(* POU SCIT_AlarmStop, ST *)
FUNCTION_BLOCK SCIT_AlarmStop
VAR_INPUT
	NETID 			: T_AmsNetId;
	PORT 			: UINT;
	WRTRD 		: BOOL;
	TMOUT 		: TIME := DEFAULT_ADS_TIMEOUT;
END_VAR
VAR_OUTPUT
	BUSY 			: BOOL;
	ERR 			: BOOL;
	ERRID 			: UDINT;
	RESULT 			: WORD;
	ADDERRORINFO 	: WORD;
END_VAR
VAR
	ADSRDWRT1		: ADSRDWRT;
	BusyFlanke 		: F_TRIG;
	StartFlanke 	: R_TRIG;
	ReadResult 		: ReadResult_t;
END_VAR
	StartFlanke(CLK:=WRTRD );
	IF StartFlanke.Q THEN
		RESULT := 0;
		ADDERRORINFO := 0;
		ReadResult.High1 := 0;
		ReadResult.Low1 := 0;
		ReadResult.High2 := 0;
		ReadResult.Low2 := 0;
	END_IF

	ADSRDWRT1(	NETID:= NETID,
					PORT:= PORT,
					IDXGRP:= 16#00010001,
					IDXOFFS:= 16#1303,
					WRITELEN:= 0,
					READLEN:= SIZEOF(ReadResult),
					SRCADDR:= 0,
					DESTADDR:= ADR(ReadResult),
					WRTRD:= WRTRD,
					TMOUT:= TMOUT);

	BUSY := ADSRDWRT1.BUSY;
	ERR := ADSRDWRT1.ERR;
	ERRID := ADSRDWRT1.ERRID;

	BusyFlanke(CLK:=BUSY);
	IF BusyFlanke.Q THEN
		RESULT := ReadResult.High1 * 256 + ReadResult.Low1;
		IF RESULT = 0 THEN
			ADDERRORINFO := 0;
		ELSE
			ADDERRORINFO := ReadResult.High2 * 256 + ReadResult.Low2;
		END_IF
	END_IF
END_FUNCTION_BLOCK

(* POU SCIT_ConfDevErrAll, ST *)
FUNCTION_BLOCK SCIT_ConfDevErrAll
VAR_INPUT
	NETID 			: T_AmsNetId;
	PORT 			: UINT;
	WRTRD 		: BOOL;
	TMOUT 		: TIME := DEFAULT_ADS_TIMEOUT;
END_VAR
VAR_OUTPUT
	BUSY 			: BOOL;
	ERR 			: BOOL;
	ERRID 			: UDINT;
	RESULT 			: WORD;
	ADDERRORINFO 	: WORD;
END_VAR
VAR
	ADSRDWRT1		: ADSRDWRT;
	BusyFlanke 		: F_TRIG;
	StartFlanke 	: R_TRIG;

	ReadResult 		: ReadResult_t;
	WriteData 		: DWORD;
END_VAR
	StartFlanke(CLK:=WRTRD );
	IF StartFlanke.Q THEN
		RESULT := 0;
		ADDERRORINFO := 0;
		ReadResult.High1 := 0;
		ReadResult.Low1 := 0;
		ReadResult.High2 := 0;
		ReadResult.Low2 := 0;
		WriteData := 16#00000400;
	END_IF

	ADSRDWRT1(	NETID:= NETID,
					PORT:= PORT,
					IDXGRP:= 16#00010001,
					IDXOFFS:= 16#0714,
					WRITELEN:= SIZEOF(WriteData),
					READLEN:= SIZEOF(ReadResult),
					SRCADDR:= ADR(WriteData),
					DESTADDR:= ADR(ReadResult),
					WRTRD:= WRTRD,
					TMOUT:= TMOUT);

	BUSY := ADSRDWRT1.BUSY;
	ERR := ADSRDWRT1.ERR;
	ERRID := ADSRDWRT1.ERRID;

	BusyFlanke(CLK:=BUSY);
	IF BusyFlanke.Q THEN
		RESULT := ReadResult.High1 * 256 + ReadResult.Low1;
		IF RESULT = 0 THEN
			ADDERRORINFO := 0;
		ELSE
			ADDERRORINFO := ReadResult.High2 * 256 + ReadResult.Low2;
		END_IF
	END_IF
END_FUNCTION_BLOCK

(* POU SCIT_ControlActiveConfiguration, ST *)
FUNCTION_BLOCK SCIT_ControlActiveConfiguration
VAR_INPUT
	NETID 			: T_AmsNetId;
	PORT 			: UINT;
	WRTRD 			: BOOL;
	TMOUT 			: TIME := DEFAULT_ADS_TIMEOUT;
	SWITCH_CODE 	: WORD;
	DEVICE_NO 		: WORD;
END_VAR
VAR_OUTPUT
	BUSY 			: BOOL;
	ERR 			: BOOL;
	ERRID 			: UDINT;
	RESULT 			: WORD;
	ADDERRORINFO 	: WORD;
END_VAR
VAR
	ADSRDWRT1		: ADSRDWRT;
	BusyFlanke 		: F_TRIG;
	StartFlanke 	: R_TRIG;
	ReadResult 		: ReadResult_t;
	WriteData 		: ControlActiveConfiguration_t;
END_VAR
	StartFlanke(CLK:=WRTRD );
	IF StartFlanke.Q THEN
		RESULT := 0;
		ADDERRORINFO := 0;
		ReadResult.High1 := 0;
		ReadResult.Low1 := 0;
		ReadResult.High2 := 0;
		ReadResult.Low2 := 0;
		WriteData.HighSwitchCode := WORD_TO_BYTE(SWITCH_CODE / 256);
		WriteData.LowSwitchCode := WORD_TO_BYTE(SWITCH_CODE);
		WriteData.High1 := 0;
		WriteData.Low1 := 1;
		WriteData.HighDeviceNo := WORD_TO_BYTE(DEVICE_NO / 256);
		WriteData.LowDeviceNo := WORD_TO_BYTE(DEVICE_NO);
	END_IF

	ADSRDWRT1(	NETID:= NETID,
					PORT:= PORT,
					IDXGRP:= 16#00010001,
					IDXOFFS:= 16#0713,
					WRITELEN:= SIZEOF(WriteData),
					READLEN:= SIZEOF(ReadResult),
					SRCADDR:= ADR(WriteData),
					DESTADDR:= ADR(ReadResult),
					WRTRD:= WRTRD,
					TMOUT:= TMOUT);

	BUSY := ADSRDWRT1.BUSY;
	ERR := ADSRDWRT1.ERR;
	ERRID := ADSRDWRT1.ERRID;

	BusyFlanke(CLK:=BUSY);
	IF BusyFlanke.Q THEN
		RESULT := ReadResult.High1 * 256 + ReadResult.Low1;
		IF RESULT = 0 THEN
			ADDERRORINFO := 0;
		ELSE
			ADDERRORINFO := ReadResult.High2 * 256 + ReadResult.Low2;
		END_IF
	END_IF
END_FUNCTION_BLOCK

(* POU SCIT_DeactivateConfiguration, ST *)
FUNCTION_BLOCK SCIT_DeactivateConfiguration
VAR_INPUT
	NETID 			: T_AmsNetId;
	PORT 			: UINT;
	WRTRD 		: BOOL;
	TMOUT 		: TIME := DEFAULT_ADS_TIMEOUT;
END_VAR
VAR_OUTPUT
	BUSY 			: BOOL;
	ERR 			: BOOL;
	ERRID 			: UDINT;
	RESULT 			: WORD;
	ADDERRORINFO 	: WORD;
END_VAR
VAR
	ADSRDWRT1		: ADSRDWRT;
	BusyFlanke 		: F_TRIG;
	StartFlanke 	: R_TRIG;
	ReadResult 		: ReadResult_t;
	WriteData 		: HLword_t;
END_VAR
	StartFlanke(CLK:=WRTRD );
	IF StartFlanke.Q THEN
		RESULT := 0;
		ADDERRORINFO := 0;
		ReadResult.High1 := 0;
		ReadResult.Low1 := 0;
		ReadResult.High2 := 0;
		ReadResult.Low2 := 0;
		WriteData.High := 0;
		WriteData.Low := 1;
	END_IF

	ADSRDWRT1(	NETID:= NETID,
					PORT:= PORT,
					IDXGRP:= 16#00010001,
					IDXOFFS:= 16#0712,
					WRITELEN:= SIZEOF(WriteData),
					READLEN:= SIZEOF(ReadResult),
					SRCADDR:= ADR(WriteData),
					DESTADDR:= ADR(ReadResult),
					WRTRD:= WRTRD,
					TMOUT:= TMOUT);

	BUSY := ADSRDWRT1.BUSY;
	ERR := ADSRDWRT1.ERR;
	ERRID := ADSRDWRT1.ERRID;

	BusyFlanke(CLK:=BUSY);
	IF BusyFlanke.Q THEN
		RESULT := ReadResult.High1 * 256 + ReadResult.Low1;
		IF RESULT = 0 THEN
			ADDERRORINFO := 0;
		ELSE
			ADDERRORINFO := ReadResult.High2 * 256 + ReadResult.Low2;
		END_IF
	END_IF
END_FUNCTION_BLOCK

(* POU SCIT_GetErrorInfo, ST *)
FUNCTION_BLOCK SCIT_GetErrorInfo
VAR_INPUT
	NETID 			: T_AmsNetId;
	PORT 			: UINT;
	WRTRD 		: BOOL;
	TMOUT 		: TIME := DEFAULT_ADS_TIMEOUT;
END_VAR
VAR_OUTPUT
	BUSY 			: BOOL;
	ERR 			: BOOL;
	ERRID 			: UDINT;
	RESULT 			: WORD;
	ERRORCODE 		: WORD;
	ADDERRORINFO 	: WORD;
END_VAR
VAR
	ADSRDWRT1		: ADSRDWRT;
	BusyFlanke 		: F_TRIG;
	StartFlanke 	: R_TRIG;
	WriteData 		: HLword_t;
	ReadResult 		: GetErrorInfo_t;
END_VAR
	StartFlanke(CLK:=WRTRD );
	IF StartFlanke.Q THEN
		RESULT := 0;
		ERRORCODE := 0;
		ADDERRORINFO := 0;
		ReadResult.HighResult := 0;
		ReadResult.LowResult := 0;
		ReadResult.HighEntryCount := 0;
		ReadResult.LowEntryCount := 0;
		ReadResult.HighErrorCode := 0;
		ReadResult.LowErrorCode := 0;
		ReadResult.HighAddErrInfo := 0;
		ReadResult.LowAddErrInfo := 0;

		WriteData.High := 0;
		WriteData.Low := 0;
	END_IF

	ADSRDWRT1(	NETID:= NETID,
					PORT:= PORT,
					IDXGRP:= 16#00010001,
					IDXOFFS:= 16#0316,
					WRITELEN:= 0,
					READLEN:= SIZEOF(ReadResult),
					SRCADDR:= ADR(WriteData),
					DESTADDR:= ADR(ReadResult),
					WRTRD:= WRTRD,
					TMOUT:= TMOUT);

	BUSY := ADSRDWRT1.BUSY;
	ERR := ADSRDWRT1.ERR;
	ERRID := ADSRDWRT1.ERRID;

	BusyFlanke(CLK:=BUSY);
	IF BusyFlanke.Q THEN
		RESULT := ReadResult.HighResult * 256 + ReadResult.LowResult;
		ERRORCODE := ReadResult.HighErrorCode * 256 + ReadResult.LowErrorCode;
		ADDERRORINFO := ReadResult.HighAddErrInfo * 256 + ReadResult.LowAddErrInfo;
	END_IF
END_FUNCTION_BLOCK

(* POU SCIT_StartDataTransfer, ST *)
FUNCTION_BLOCK SCIT_StartDataTransfer
VAR_INPUT
	NETID 			: T_AmsNetId;
	PORT 			: UINT;
	WRTRD 		: BOOL;
	TMOUT 		: TIME := DEFAULT_ADS_TIMEOUT;
END_VAR
VAR_OUTPUT
	BUSY 			: BOOL;
	ERR 			: BOOL;
	ERRID 			: UDINT;
	RESULT 			: WORD;
	ADDERRORINFO 	: WORD;
END_VAR
VAR
	ADSRDWRT1		: ADSRDWRT;
	BusyFlanke 		: F_TRIG;
	StartFlanke 	: R_TRIG;
	ReadResult 		: ReadResult_t;
END_VAR
	StartFlanke(CLK:=WRTRD );
	IF StartFlanke.Q THEN
		RESULT := 0;
		ADDERRORINFO := 0;
		ReadResult.High1 := 0;
		ReadResult.Low1 := 0;
		ReadResult.High2 := 0;
		ReadResult.Low2 := 0;
	END_IF

	ADSRDWRT1(	NETID:= NETID,
					PORT:= PORT,
					IDXGRP:= 16#00010001,
					IDXOFFS:= 16#0701,
					WRITELEN:= 0,
					READLEN:= SIZEOF(ReadResult),
					SRCADDR:= 0,
					DESTADDR:= ADR(ReadResult),
					WRTRD:= WRTRD,
					TMOUT:= TMOUT);

	BUSY := ADSRDWRT1.BUSY;
	ERR := ADSRDWRT1.ERR;
	ERRID := ADSRDWRT1.ERRID;

	BusyFlanke(CLK:=BUSY);
	IF BusyFlanke.Q THEN
		RESULT := ReadResult.High1 * 256 + ReadResult.Low1;
		IF RESULT = 0 THEN
			ADDERRORINFO := 0;
		ELSE
			ADDERRORINFO := ReadResult.High2 * 256 + ReadResult.Low2;
		END_IF
	END_IF
END_FUNCTION_BLOCK

(* POU SCIT_StopDataTransfer, ST *)
FUNCTION_BLOCK SCIT_StopDataTransfer
VAR_INPUT
	NETID 			: T_AmsNetId;
	PORT 			: UINT;
	WRTRD 		: BOOL;
	TMOUT 		: TIME := DEFAULT_ADS_TIMEOUT;
END_VAR
VAR_OUTPUT
	BUSY 			: BOOL;
	ERR 			: BOOL;
	ERRID 			: UDINT;
	RESULT 			: WORD;
	ADDERRORINFO 	: WORD;
END_VAR
VAR
	ADSRDWRT1		: ADSRDWRT;
	BusyFlanke 		: F_TRIG;
	StartFlanke 	: R_TRIG;
	ReadResult 		: ReadResult_t;
	WriteData 		: WORD;
END_VAR
	StartFlanke(CLK:=WRTRD );
	IF StartFlanke.Q THEN
		RESULT := 0;
		ADDERRORINFO := 0;
		ReadResult.High1 := 0;
		ReadResult.Low1 := 0;
		ReadResult.High2 := 0;
		ReadResult.Low2 := 0;
		WriteData := 0;
	END_IF

	ADSRDWRT1(	NETID:= NETID,
					PORT:= PORT,
					IDXGRP:= 16#00010001,
					IDXOFFS:= 16#0702,
					WRITELEN:= SIZEOF(WriteData),
					READLEN:= SIZEOF(ReadResult),
					SRCADDR:= ADR(WriteData),
					DESTADDR:= ADR(ReadResult),
					WRTRD:= WRTRD,
					TMOUT:= TMOUT);

	BUSY := ADSRDWRT1.BUSY;
	ERR := ADSRDWRT1.ERR;
	ERRID := ADSRDWRT1.ERRID;

	BusyFlanke(CLK:=BUSY);
	IF BusyFlanke.Q THEN
		RESULT := ReadResult.High1 * 256 + ReadResult.Low1;
		IF RESULT = 0 THEN
			ADDERRORINFO := 0;
		ELSE
			ADDERRORINFO := ReadResult.High2 * 256 + ReadResult.Low2;
		END_IF
	END_IF
END_FUNCTION_BLOCK
